{attribute 'qualified_only'}
{attribute 'strict'}
TYPE eStopMode :
(
    ControlledStop := 1,
    StopAndDisable := 2
);
END_TYPE

(* stored: Version 1.1.0.1, ProductVersion 3.1.4026.18
   DUT eStopMode: Id {d246b69f-46fc-4a3b-9bc0-f1d88280210e} *)
